// TIA Portal V17 program export: 1 tag tables, 0 data types, 0 data blocks, 5 code blocks (in call order from the OBs), 1 instance data blocks

VAR_GLOBAL   // PLC tag table "Default tag table"
   Sw1 AT %I0.0 : Bool;
   Sw2 AT %I0.1 : Bool;
   Output1 AT %Q0.0 : Bool;
   Output2 AT %Q0.1 : Bool;
   Sw3 AT %I0.2 : Bool;
   Sw4 AT %I0.3 : Bool;
   Sw5 AT %I0.4 : Bool;
   Sw6 AT %I0.5 : Bool;
   Sw7 AT %I0.6 : Bool;
   Sw8 AT %I0.7 : Bool;
   Sw9 AT %I1.0 : Bool;
   Sw10 AT %I1.1 : Bool;
   Output3 AT %Q0.2 : Bool;
   Output4 AT %Q0.3 : Bool;
   Output6 AT %Q0.5 : Bool;
   Sw11 AT %I1.2 : Bool;
   Sw12 AT %I1.3 : Bool;
   Output12 AT %Q0.7 : Bool;
   Output11 AT %Q0.6 : Bool;
END_VAR

ORGANIZATION_BLOCK "Main"   // OB1, LAD, ProgramCycle
TITLE = "Main Program Sweep (Cycle)"
{ S7_Optimized_Access := 'TRUE' }
VERSION : 0.1
// stored: AutoNumber true, IsIECCheckEnabled false, SetENOAutomatically false
   VAR_INPUT
      Initial_Call : Bool;   // Initial call of this OB
      Remanence : Bool;   // =True, if remanent data are available
   END_VAR
BEGIN

REGION Network 1
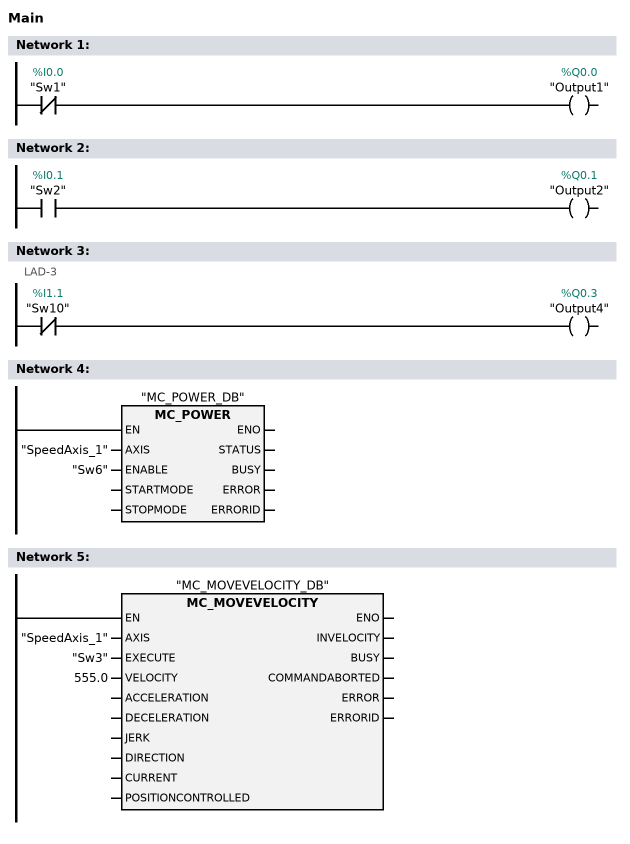
   RUNG wire#powerrail
      I_Contact( "Sw1" )
      Coil( "Output1" )
   END_RUNG
   // the same network as SCL:
   "Output1" := NOT "Sw1";
END_REGION

REGION Network 2
   RUNG wire#powerrail
      Contact( "Sw2" )
      Coil( "Output2" )
   END_RUNG
   // the same network as SCL:
   "Output2" := "Sw2";
END_REGION

REGION Network 3
   // LAD-3
   RUNG wire#powerrail
      I_Contact( "Sw10" )
      Coil( "Output4" )
   END_RUNG
   // the same network as SCL:
   "Output4" := NOT "Sw10";
END_REGION

REGION Network 4
   RUNG wire#powerrail
      "MC_POWER_DB".MC_POWER(Axis := "SpeedAxis_1", Enable := "Sw6", StartMode :=, StopMode :=, Status =>, Busy =>, Error =>, ErrorId =>)
   END_RUNG
   // the same network as SCL:
   "MC_POWER_DB"(Axis := "SpeedAxis_1", Enable := "Sw6");   // MC_POWER
END_REGION

REGION Network 5
   RUNG wire#powerrail
      "MC_MOVEVELOCITY_DB".MC_MOVEVELOCITY(Axis := "SpeedAxis_1", Execute := "Sw3", Velocity := 555.0, Acceleration :=, Deceleration :=, Jerk :=, Direction :=, Current :=, PositionControlled :=, InVelocity =>, Busy =>, CommandAborted =>, Error =>, ErrorId =>)
   END_RUNG
   // the same network as SCL:
   "MC_MOVEVELOCITY_DB"(Axis := "SpeedAxis_1", Execute := "Sw3", Velocity := 555.0);   // MC_MOVEVELOCITY
END_REGION
END_ORGANIZATION_BLOCK

FUNCTION_BLOCK "Main_Safety_RTG1"   // FB1, F_FBD
{ S7_Optimized_Access := 'TRUE' }
VERSION : 0.1
// stored: AutoNumber false, IsIECCheckEnabled false, UDAEnableTagReadback false
BEGIN
END_FUNCTION_BLOCK

FUNCTION "Routine_1" : Void   // FC2, LAD
{ S7_Optimized_Access := 'TRUE' }
VERSION : 0.1
// stored: AutoNumber true, IsIECCheckEnabled false, SetENOAutomatically false, UDAEnableTagReadback false
BEGIN

REGION Network 1
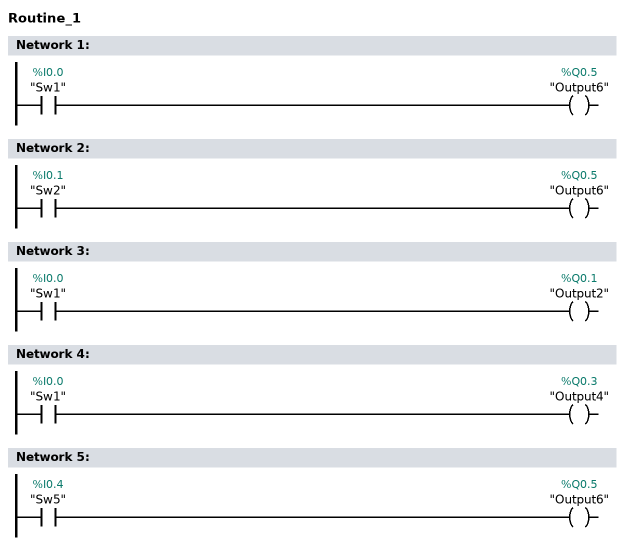
   RUNG wire#powerrail
      Contact( "Sw1" )
      Coil( "Output6" )
   END_RUNG
   // the same network as SCL:
   "Output6" := "Sw1";
END_REGION

REGION Network 2
   RUNG wire#powerrail
      Contact( "Sw2" )
      Coil( "Output6" )
   END_RUNG
   // the same network as SCL:
   "Output6" := "Sw2";
END_REGION

REGION Network 3
   RUNG wire#powerrail
      Contact( "Sw1" )
      Coil( "Output2" )
   END_RUNG
   // the same network as SCL:
   "Output2" := "Sw1";
END_REGION

REGION Network 4
   RUNG wire#powerrail
      Contact( "Sw1" )
      Coil( "Output4" )
   END_RUNG
   // the same network as SCL:
   "Output4" := "Sw1";
END_REGION

REGION Network 5
   RUNG wire#powerrail
      Contact( "Sw5" )
      Coil( "Output6" )
   END_RUNG
   // the same network as SCL:
   "Output6" := "Sw5";
END_REGION
END_FUNCTION

FUNCTION "Routine_2" : Void   // FC1, LAD
{ S7_Optimized_Access := 'TRUE' }
VERSION : 0.1
// stored: AutoNumber true, IsIECCheckEnabled false, SetENOAutomatically false, UDAEnableTagReadback false
BEGIN

REGION Network 1
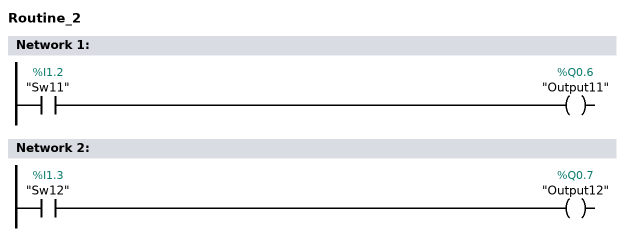
   RUNG wire#powerrail
      Contact( "Sw11" )
      Coil( "Output11" )
   END_RUNG
   // the same network as SCL:
   "Output11" := "Sw11";
END_REGION

REGION Network 2
   RUNG wire#powerrail
      Contact( "Sw12" )
      Coil( "Output12" )
   END_RUNG
   // the same network as SCL:
   "Output12" := "Sw12";
END_REGION
END_FUNCTION

FUNCTION "Routine_3" : Void   // FC3, LAD
{ S7_Optimized_Access := 'TRUE' }
VERSION : 0.1
// stored: AutoNumber true, IsIECCheckEnabled false, SetENOAutomatically false, UDAEnableTagReadback false
BEGIN

REGION Network 1
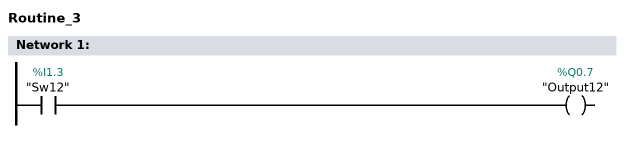
   RUNG wire#powerrail
      Contact( "Sw12" )
      Coil( "Output12" )
   END_RUNG
   // the same network as SCL:
   "Output12" := "Sw12";
END_REGION
END_FUNCTION

DATA_BLOCK "Main_Safety_RTG1_DB"   // DB1, F_DB
NAME : FUSI
VERSION : 0.1
// stored: AutoNumber true, InstanceOfName Main_Safety_RTG1, InstanceOfType FB
"Main_Safety_RTG1"
BEGIN
END_DATA_BLOCK
